{attribute 'reflection'}
FUNCTION_BLOCK ABSTRACT Objective IMPLEMENTS iObjective
VAR_INPUT
END_VAR
VAR
	
	TrackedMovers		: ARRAY [0..GVL.NUM_MOVERS-1] OF POINTER TO Mover;
	TrackedMoverCount	: UINT;	

END_VAR
VAR_OUTPUT
		
	{attribute 'instance-path'}
	{attribute 'noinit'}
	InstancePath		: STRING;		// Unique variable path of the instance
	
END_VAR


PROPERTY CurrentMover : Reference TO Mover
GET
END_GET
SET
END_SET
END_PROPERTY

METHOD RegisterMover : BOOL
VAR_INPUT	
	// NewMover		: POINTER TO Mover;
	NewMover		: REFERENCE TO Mover;
	
END_VAR

VAR
	i				: USINT;
	duplicateFound	: BOOL;
	emptyIDX		: USINT;
END_VAR

(*
	Add a mover to a list of movers tracked by the objective.
	Movers can't be added multiple times, so check for duplicates
	Movers can't overwrite others in the list, so check that the array element is clear
*)

//IF NewMover <> 0 THEN				// validate pointer

IF __ISVALIDREF( NewMover ) THEN	// validate alias
	
	duplicateFound		:= FALSE;		// default to false, counterexample below
	TrackedMoverCount	:= 0;			// reset to zero, incremented below

	FOR i := 0 TO SIZEOF(TrackedMovers)/SIZEOF(TrackedMovers[i])-1 DO
		IF TrackedMovers[i] <> 0 THEN			
			IF ADR(NewMover) = TrackedMovers[i] THEN
				duplicateFound	:= TRUE;				// this mover already tracked
			END_IF			
			TrackedMoverCount	:= TrackedMoverCount + 1;
		ELSE
			emptyIDX			:= i;					// confirmed open array element
		END_IF
	END_FOR

	IF duplicateFound = FALSE THEN
		TrackedMovers[emptyIDX]		:= ADR( NewMover );		// new mover goes into open array element
		TrackedMoverCount			:= TrackedMoverCount + 1;
	END_IF

ELSE
	ADSLOGSTR(ADSLOG_MSGTYPE_LOG,'Error: Mover input is invalid','');
END_IF
END_METHOD

METHOD UnregisterCurrent : BOOL
VAR_INPUT
END_VAR


THIS^.UnregisterMover(CurrentMover);
END_METHOD

METHOD UnregisterMover : BOOL
VAR_INPUT
	// RemovingMover		: POINTER TO Mover;
	RemovingMover		: REFERENCE TO Mover;
END_VAR
VAR
	i					: USINT;
	duplicateFound		: BOOL;
END_VAR


(*
	Remove a mover to a list of movers tracked by the objective.
	Only movers in the list can be removed, otherwise nothing happens
*)


// IF RemovingMover <> 0 THEN			// validate pointer
IF __ISVALIDREF( RemovingMover ) THEN
	
	TrackedMoverCount	:= 0;
	
	FOR i := 0 TO SIZEOF( TrackedMovers )/SIZEOF( TrackedMovers[0] )-1 DO
		IF TrackedMovers[i] <> 0 THEN	// validate pointer
					
			TrackedMoverCount		:= TrackedMoverCount + 1;
			
			IF ADR(RemovingMover) = TrackedMovers[i] THEN
				TrackedMovers[i]	:= 0;		// remove the pointer
				TrackedMoverCount	:= TrackedMoverCount - 1;
			END_IF
		
		END_IF
	END_FOR

ELSE
	ADSLOGSTR(ADSLOG_MSGTYPE_LOG,'Error: Mover input is invalid','');
END_IF
END_METHOD

END_FUNCTION_BLOCK

(* stored: Version 1.1.0.1, ProductVersion 3.1.4024.9
   POU Objective: Id {72371872-54aa-4f25-a82d-ba585015a7c5}, SpecialFunc None
   Property CurrentMover: Id {be94617c-1fc3-4981-a1c2-c43a4094d43b}
   Get Get: Id {12bc2a84-bf29-43b6-b2d1-79d6711b1b04}
   Set Set: Id {a537d59c-ece5-4c34-bc20-58aad19c2d06}
   Method RegisterMover: Id {8354cf16-6187-4fe4-976a-42e2fe3b8399}
   Method UnregisterCurrent: Id {8c43e469-bfcf-4444-8690-ba524026657d}
   Method UnregisterMover: Id {18c8f6fd-1567-45b0-85d6-dc2464792b83} *)
